FUNCTION_BLOCK DINT_Param
VAR_INPUT PERSISTENT
	val			: DINT;
END_VAR

END_FUNCTION_BLOCK

(* stored: Version 1.1.0.1
   POU DINT_Param: Id {a2596563-098b-48b4-a34e-539eec843427}, SpecialFunc None *)
